FUNCTION_BLOCK FB_SystemTime
VAR_INPUT
END_VAR
VAR_OUTPUT
END_VAR
VAR
	GetLocalSystemTime 	: FB_LocalSystemTime;
	wDateW				: WORD;
END_VAR

GetLocalSystemTime(bEnable := TRUE);

PROPERTY dtDateTimeFull : DT
GET
dtDateTimeFull 	:= SYSTEMTIME_TO_DT(GetLocalSystemTime.systemTime);
END_GET
END_PROPERTY

PROPERTY sDate : STRING
GET
sDate	:= MID(sDateTimeFull,10,1);
END_GET
END_PROPERTY

PROPERTY sDateTime : STRING
GET
sDateTime := MID(sDateTimeFull,19,1);
END_GET
END_PROPERTY

PROPERTY sDateTimeFull : STRING
GET
sDateTimeFull 	:= SYSTEMTIME_TO_STRING(GetLocalSystemTime.systemTime);
END_GET
END_PROPERTY

PROPERTY sDayOfWeek : STRING
GET
wDateW	:=  GetLocalSystemTime.systemTime.wDayOfWeek;
IF wDateW = 0 THEN
	sDayOfWeek := 'Sunday';
ELSIF wDateW = 1 THEN
	sDayOfWeek := 'Monday';
ELSIF wDateW = 2 THEN
	sDayOfWeek := 'Tuesday';
ELSIF wDateW = 3 THEN
	sDayOfWeek := 'Wednesday';
ELSIF wDateW = 4 THEN
	sDayOfWeek := 'Thursday';
ELSIF wDateW = 5 THEN
	sDayOfWeek := 'Friday';
ELSIF wDateW = 6 THEN
	sDayOfWeek := 'Saturday';
END_IF
END_GET
END_PROPERTY

PROPERTY sTime : STRING
GET
sTime := MID(sDateTimeFull,8,12);
END_GET
END_PROPERTY

PROPERTY wDay : Word
GET
wDay :=  GetLocalSystemTime.systemTime.wDay;
END_GET
END_PROPERTY

PROPERTY wHour : WORD
GET
wHour	:=	GetLocalSystemTime.systemTime.wHour;
END_GET
END_PROPERTY

PROPERTY wMilliSeconds : WORD
GET
wMilliseconds	:=	GetLocalSystemTime.systemTime.wMilliseconds;
END_GET
END_PROPERTY

PROPERTY wMinute : WORD
GET
wMinute	:=	GetLocalSystemTime.systemTime.wMinute;
END_GET
END_PROPERTY

PROPERTY wMonth : Word
GET
wMonth	:=  GetLocalSystemTime.systemTime.wMonth;
END_GET
END_PROPERTY

PROPERTY wSecond : WORD
GET
wSecond	:=	GetLocalSystemTime.systemTime.wSecond;
END_GET
END_PROPERTY

PROPERTY wYear : Word
GET
wYear :=  GetLocalSystemTime.systemTime.wYear;
END_GET
END_PROPERTY

END_FUNCTION_BLOCK

(* stored: Version 1.1.0.1, ProductVersion 3.1.4024.12
   POU FB_SystemTime: Id {2c748e60-9fff-4e65-a896-a31986ab9309}, SpecialFunc None
   Property dtDateTimeFull: Id {5d9db981-e399-476f-9f44-b7969859fd33}
   Get Get: Id {68209983-270f-4891-9dce-ea500a943a8e}
   Property sDate: Id {adb2b91a-c3a4-4948-a9ab-17c03886c6a1}
   Get Get: Id {356267ce-a5ea-4b87-99e8-11910f8c4ecc}
   Property sDateTime: Id {ddd67e66-e1a4-4207-aac8-28653586b9f3}
   Get Get: Id {e6044f6a-3395-4669-a1fa-a4abfda6bc18}
   Property sDateTimeFull: Id {ec972ccc-929a-446b-93da-990283db8464}
   Get Get: Id {f58ef226-2140-466f-b534-95dc853dde3e}
   Property sDayOfWeek: Id {a30c2e4c-1ca2-4e89-9e2d-02cd951dbf57}
   Get Get: Id {33e404d2-2ba9-4b57-92a7-89c7b51daf56}
   Property sTime: Id {dc607d9d-5fbb-4395-9f68-3f6b3c933e1d}
   Get Get: Id {a44799e2-26a8-4375-9f32-6f7d6032d943}
   Property wDay: Id {0509d925-5e29-455a-a44b-917daa4ddc34}
   Get Get: Id {dc6ac976-79de-40ca-ad36-9b363cffc2be}
   Property wHour: Id {14568886-a968-428a-89a9-3c243eca2652}
   Get Get: Id {8a383dfd-47d5-41e3-a0a4-8bb82b88254c}
   Property wMilliSeconds: Id {f711972c-4a15-43a3-ad14-70806eb762d2}
   Get Get: Id {fee1178b-5cb3-41fa-8541-9d654f923b18}
   Property wMinute: Id {ac2d1731-3055-4d58-aa2f-70efe444c3ed}
   Get Get: Id {ffb7fc96-817c-4af1-b070-c2026c0c9ed3}
   Property wMonth: Id {b5c40313-975b-4dad-895d-5f967944c06e}
   Get Get: Id {b4e49317-a551-4f67-9692-0ea9e1b429e7}
   Property wSecond: Id {942dd1c0-a6e6-4375-8dd6-b31d1974723f}
   Get Get: Id {6393d2f1-5906-4562-82d1-05cbacc402d7}
   Property wYear: Id {1e665b64-e124-4d08-81b7-d54481c382a4}
   Get Get: Id {feda2073-6e29-4570-875c-38ef9ac368fa} *)
